FUNCTION_BLOCK ABSTRACT CyclicBase IMPLEMENTS ICyclic
VAR
END_VAR

METHOD PUBLIC ABSTRACT Cycle : BOOL
VAR_INPUT
END_VAR
END_METHOD

END_FUNCTION_BLOCK

(* stored: Version 1.1.0.1, ProductVersion 3.1.4024.12
   POU CyclicBase: Id {822a4270-a76d-44ce-8055-ee2099020175}, SpecialFunc None
   Method Cycle: Id {9762b721-7f92-40df-8e44-4acdbac204f1} *)
